TYPE stProductInfo :
	STRUCT
		ProductName				: STRING;
		BarcodeReference		: STRING;
		EANVariant				: STRING;
		LinkUpSource			: STRING;
		CodeVariant				: STRING;
		ProductLength			: UINT;
		ProductWidth			: UINT;
		ProductHeight			: UINT;
		ProductPattern			: USINT;
		Stacking				: UINT;
		OffsetPattern			: stCustomPattern;
	END_STRUCT
END_TYPE

(* stored: Version 1.1.0.1, ProductVersion 3.1.4024.6
   DUT stProductInfo: Id {579b996e-03d0-4615-a4d9-ea99f873d955} *)
